// TIA Portal V15.1 export
// export: Created 2020-06-12T07:35:48.5224609Z, ExportSetting None, DisplayName Totally Integrated Automation Portal, DisplayVersion V15.1, DisplayName TIA Portal Openness, DisplayVersion V15.1, DisplayName STEP 7 Professional, DisplayVersion V15.1, DisplayName STEP 7 Safety, DisplayVersion V15.1, DisplayName WinCC Advanced, DisplayVersion V15.1
FUNCTION "PWR_trafo" : Void   // FC143, FBD
TITLE = Transformer with a vareing secondary voltage
{ S7_Optimized_Access := 'TRUE' }
// stored: SetENOAutomatically False
   VAR_TEMP
      tContEn : Bool;
      tContEnS : Bool;
      tContOn : Bool;
      tContLock : Bool;
      tContLStop : Bool;
      tContLSbot : Bool;
      tContCbOn : Bool;
      tContOnInc : Bool;
      tContOnDec : Bool;
      tContRunUp : Bool;
      tContRunDown : Bool;
      tOCTReq : Bool;
      tContMode : Int;
      tContSet : Real;   // Manipulation speed (cont K)
      tContFbSet : Real;
      tContUest : Real;   // Filtered actual voltage (filter K)
      tContUestS : Real;   // Filtered actual voltage (filter S)
      tContUact : Real;   // Unfiltered measured voltage
      tContUset : Real;   // Target voltage
      tContUmin : Real;   // Minimal voltage (w/o load)
      tContUmax : Real;   // Maximal voltage (w/o load)
      tContSmax : Real;   // Maximal speed setpoint
      tContSmin : Real;   // Minimal speed setpoint
      tContCycle : Time;
      tResult : Word;
      tTrafoCoolFault : Bool;
      tDirectOp : Bool;
      tTrdPosErr : LReal;
      tWindsPosErr : Real;
      tContIact : Real;
      tConMeasMode : Bool;
      tContUdrop : Real;
      tPosInv : Real;
      tContTgtReached : Bool;
      tXinternal : Real;
      tUload : Real;
      tIload : Real;
      tContUdrop2 : Real;
      tRbase : Real;
      tPosValid : Bool;
   END_VAR
BEGIN

REGION Network 1: Transformar is cooling
   // These signals are inverted
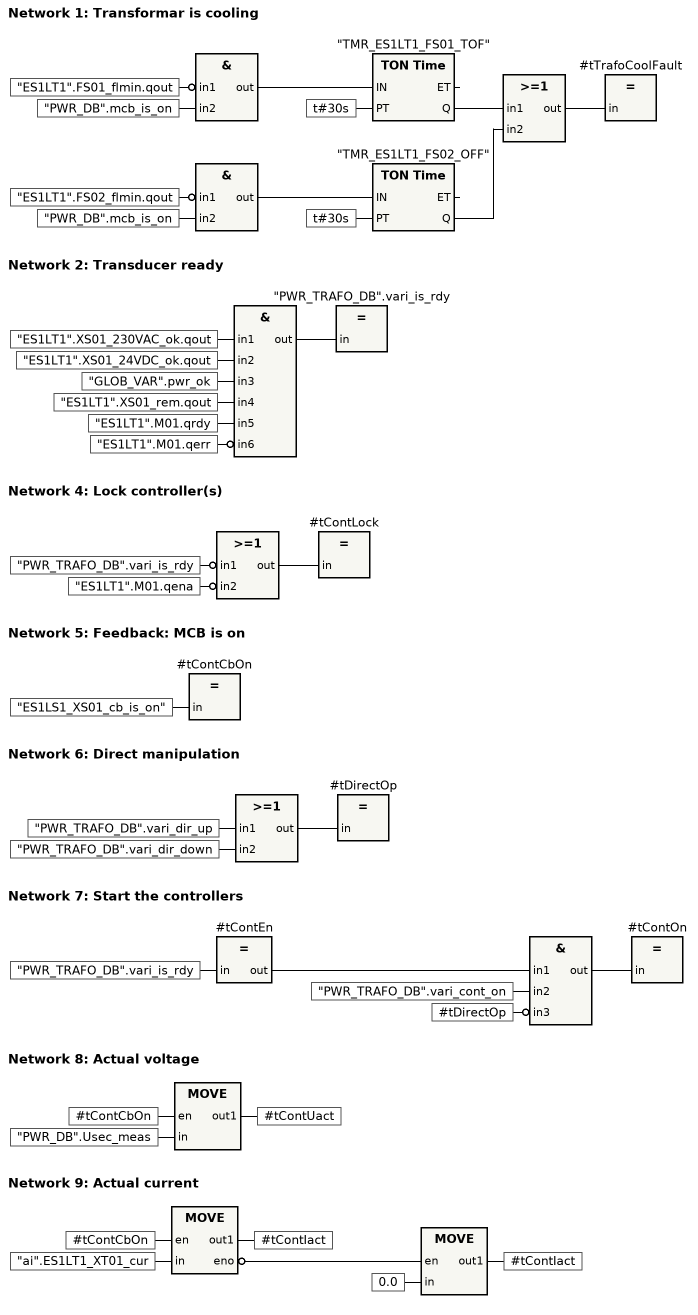
   "TMR_ES1LT1_FS01_TOF".TON(IN := NOT "ES1LT1".FS01_flmin.qout AND "PWR_DB".mcb_is_on, PT := t#30s);
   "TMR_ES1LT1_FS02_OFF".TON(IN := NOT "ES1LT1".FS02_flmin.qout AND "PWR_DB".mcb_is_on, PT := t#30s);
   #tTrafoCoolFault := "TMR_ES1LT1_FS01_TOF".Q OR "TMR_ES1LT1_FS02_OFF".Q;
END_REGION

REGION Network 2: Transducer ready
   "PWR_TRAFO_DB".vari_is_rdy := "ES1LT1".XS01_230VAC_ok.qout AND "ES1LT1".XS01_24VDC_ok.qout AND "GLOB_VAR".pwr_ok AND "ES1LT1".XS01_rem.qout AND "ES1LT1".M01.qrdy AND NOT "ES1LT1".M01.qerr;
END_REGION

REGION Network 3: -----------------------------------------------------------------------------
END_REGION

REGION Network 4: Lock controller(s)
   #tContLock := NOT "PWR_TRAFO_DB".vari_is_rdy OR NOT "ES1LT1".M01.qena;
END_REGION

REGION Network 5: Feedback: MCB is on
   #tContCbOn := "ES1LS1_XS01_cb_is_on";
END_REGION

REGION Network 6: Direct manipulation
   #tDirectOp := "PWR_TRAFO_DB".vari_dir_up OR "PWR_TRAFO_DB".vari_dir_down;
END_REGION

REGION Network 7: Start the controllers
   #tContEn := "PWR_TRAFO_DB".vari_is_rdy;
   #tContOn := "PWR_TRAFO_DB".vari_is_rdy AND "PWR_TRAFO_DB".vari_cont_on AND NOT #tDirectOp;
END_REGION

REGION Network 8: Actual voltage
   // I use these recalculation to avoid double model of voltage
   IF #tContCbOn THEN #tContUact := "PWR_DB".Usec_meas; END_IF;
END_REGION

REGION Network 9: Actual current
   IF #tContCbOn THEN #tContIact := "ai".ES1LT1_XT01_cur; END_IF;
   IF NOT #tContCbOn THEN #tContIact := 0.0; END_IF;
END_REGION

REGION Network 10: Measurement mode
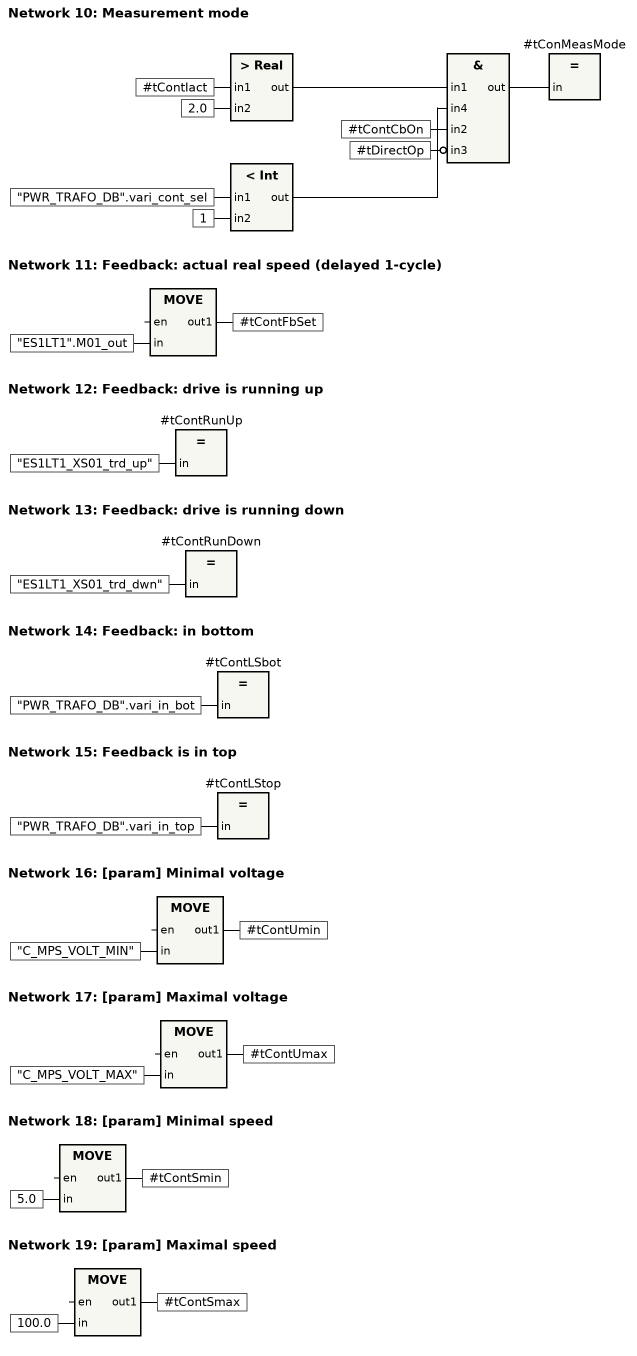
   #tConMeasMode := (#tContIact > 2.0) AND ("PWR_TRAFO_DB".vari_cont_sel < 1) AND #tContCbOn AND NOT #tDirectOp;
END_REGION

REGION Network 11: Feedback: actual real speed (delayed 1-cycle)
   #tContFbSet := "ES1LT1".M01_out;
END_REGION

REGION Network 12: Feedback: drive is running up
   #tContRunUp := "ES1LT1_XS01_trd_up";
END_REGION

REGION Network 13: Feedback: drive is running down
   #tContRunDown := "ES1LT1_XS01_trd_dwn";
END_REGION

REGION Network 14: Feedback: in bottom
   #tContLSbot := "PWR_TRAFO_DB".vari_in_bot;
END_REGION

REGION Network 15: Feedback is in top
   #tContLStop := "PWR_TRAFO_DB".vari_in_top;
END_REGION

REGION Network 16: [param] Minimal voltage
   #tContUmin := "C_MPS_VOLT_MIN";
END_REGION

REGION Network 17: [param] Maximal voltage
   #tContUmax := "C_MPS_VOLT_MAX";
END_REGION

REGION Network 18: [param] Minimal speed
   #tContSmin := 5.0;
END_REGION

REGION Network 19: [param] Maximal speed
   #tContSmax := 100.0;
END_REGION

REGION Network 20: [param] Cycle time
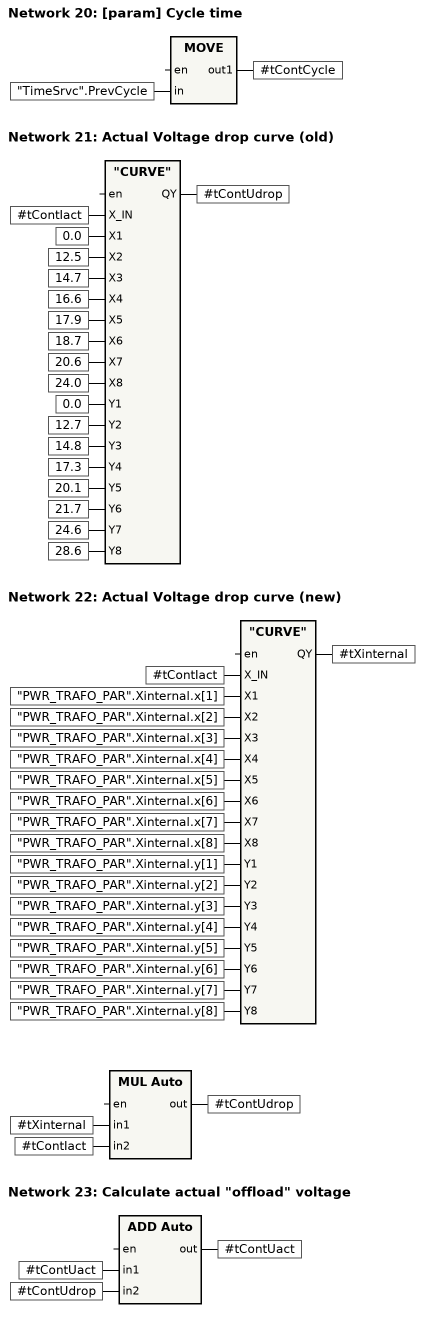
   #tContCycle := "TimeSrvc".PrevCycle;
END_REGION

REGION Network 21: Actual Voltage drop curve (old)
   // WARNING! After updating of the curve, you MUST update also the curve in the block FC "MELT_CPF_VP"
   "CURVE"(X_IN := #tContIact,
           X1 := 0.0,
           X2 := 12.5,
           X3 := 14.7,
           X4 := 16.6,
           X5 := 17.9,
           X6 := 18.7,
           X7 := 20.6,
           X8 := 24.0,
           Y1 := 0.0,
           Y2 := 12.7,
           Y3 := 14.8,
           Y4 := 17.3,
           Y5 := 20.1,
           Y6 := 21.7,
           Y7 := 24.6,
           Y8 := 28.6,
           QY => #tContUdrop);
END_REGION

REGION Network 22: Actual Voltage drop curve (new)
   // WARNING! After updating of the curve, you MUST update also the curve in the block FC "MELT_CPF_VP"
   "CURVE"(X_IN := #tContIact,
           X1 := "PWR_TRAFO_PAR".Xinternal.x[1],
           X2 := "PWR_TRAFO_PAR".Xinternal.x[2],
           X3 := "PWR_TRAFO_PAR".Xinternal.x[3],
           X4 := "PWR_TRAFO_PAR".Xinternal.x[4],
           X5 := "PWR_TRAFO_PAR".Xinternal.x[5],
           X6 := "PWR_TRAFO_PAR".Xinternal.x[6],
           X7 := "PWR_TRAFO_PAR".Xinternal.x[7],
           X8 := "PWR_TRAFO_PAR".Xinternal.x[8],
           Y1 := "PWR_TRAFO_PAR".Xinternal.y[1],
           Y2 := "PWR_TRAFO_PAR".Xinternal.y[2],
           Y3 := "PWR_TRAFO_PAR".Xinternal.y[3],
           Y4 := "PWR_TRAFO_PAR".Xinternal.y[4],
           Y5 := "PWR_TRAFO_PAR".Xinternal.y[5],
           Y6 := "PWR_TRAFO_PAR".Xinternal.y[6],
           Y7 := "PWR_TRAFO_PAR".Xinternal.y[7],
           Y8 := "PWR_TRAFO_PAR".Xinternal.y[8],
           QY => #tXinternal);
   #tContUdrop := #tXinternal * #tContIact;
END_REGION

REGION Network 23: Calculate actual "offload" voltage
   #tContUact := #tContUact + #tContUdrop;
END_REGION

REGION Network 24 (SCL): Calculate the resistance base
   IF "PWR_DB".current_flow THEN
       // I expect that this formula can do the power regulation a smooth
       #tRbase := 0.67 * "PWR_DB".Rsec_act + 0.33 * "PWR_DB".Rset;
       // but I am not sure. Well used old solution
       //#tRbase := "PWR_DB".Rsec_act;
   ELSE
       #tRbase := "PWR_DB".Rset;
   END_IF;
END_REGION

REGION Network 25: Calculate the voltage setpoint
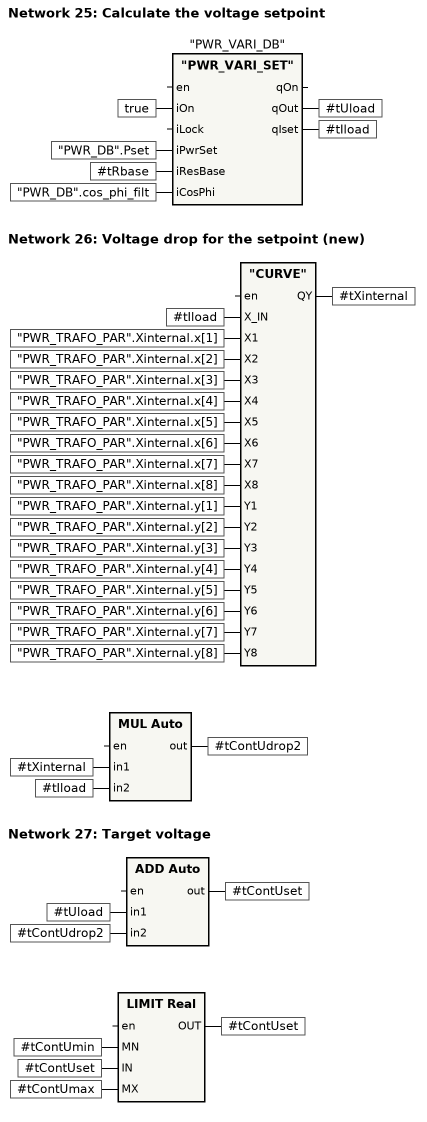
   "PWR_VARI_DB"(iOn := true,   // "PWR_VARI_SET"
                 iPwrSet := "PWR_DB".Pset,
                 iResBase := #tRbase,
                 iCosPhi := "PWR_DB".cos_phi_filt,
                 qOut => #tUload,
                 qIset => #tIload);
END_REGION

REGION Network 26: Voltage drop for the setpoint (new)
   "CURVE"(X_IN := #tIload,
           X1 := "PWR_TRAFO_PAR".Xinternal.x[1],
           X2 := "PWR_TRAFO_PAR".Xinternal.x[2],
           X3 := "PWR_TRAFO_PAR".Xinternal.x[3],
           X4 := "PWR_TRAFO_PAR".Xinternal.x[4],
           X5 := "PWR_TRAFO_PAR".Xinternal.x[5],
           X6 := "PWR_TRAFO_PAR".Xinternal.x[6],
           X7 := "PWR_TRAFO_PAR".Xinternal.x[7],
           X8 := "PWR_TRAFO_PAR".Xinternal.x[8],
           Y1 := "PWR_TRAFO_PAR".Xinternal.y[1],
           Y2 := "PWR_TRAFO_PAR".Xinternal.y[2],
           Y3 := "PWR_TRAFO_PAR".Xinternal.y[3],
           Y4 := "PWR_TRAFO_PAR".Xinternal.y[4],
           Y5 := "PWR_TRAFO_PAR".Xinternal.y[5],
           Y6 := "PWR_TRAFO_PAR".Xinternal.y[6],
           Y7 := "PWR_TRAFO_PAR".Xinternal.y[7],
           Y8 := "PWR_TRAFO_PAR".Xinternal.y[8],
           QY => #tXinternal);
   #tContUdrop2 := #tXinternal * #tIload;
END_REGION

REGION Network 27: Target voltage
   #tContUset := #tUload + #tContUdrop2;
   #tContUset := LIMIT(MN := #tContUmin, IN := #tContUset, MX := #tContUmax);
END_REGION

REGION Network 28: TRANSFORMER CONTROLLER
   // WARNING! The controler is VERY sensitive to the drive parameters
   // NOTE: 
   // - The bottom position of winds is a highest voltage
   // - The top position of winds is a lowest voltage
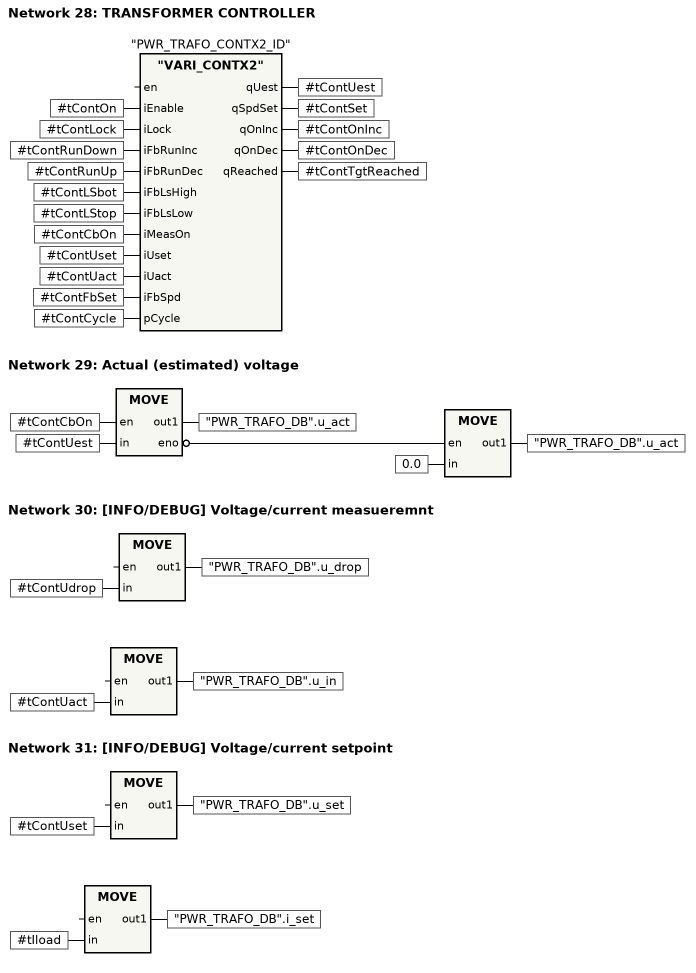
   "PWR_TRAFO_CONTX2_ID"(iEnable := #tContOn,   // "VARI_CONTX2"
                         iLock := #tContLock,
                         iFbRunInc := #tContRunDown,
                         iFbRunDec := #tContRunUp,
                         iFbLsHigh := #tContLSbot,
                         iFbLsLow := #tContLStop,
                         iMeasOn := #tContCbOn,
                         iUset := #tContUset,
                         iUact := #tContUact,
                         iFbSpd := #tContFbSet,
                         pCycle := #tContCycle,
                         qUest => #tContUest,
                         qSpdSet => #tContSet,
                         qOnInc => #tContOnInc,
                         qOnDec => #tContOnDec,
                         qReached => #tContTgtReached);
END_REGION

REGION Network 29: Actual (estimated) voltage
   IF #tContCbOn THEN "PWR_TRAFO_DB".u_act := #tContUest; END_IF;
   IF NOT #tContCbOn THEN "PWR_TRAFO_DB".u_act := 0.0; END_IF;
END_REGION

REGION Network 30: [INFO/DEBUG] Voltage/current measueremnt
   "PWR_TRAFO_DB".u_drop := #tContUdrop;
   "PWR_TRAFO_DB".u_in := #tContUact;
END_REGION

REGION Network 31: [INFO/DEBUG] Voltage/current setpoint
   "PWR_TRAFO_DB".u_set := #tContUset;
   "PWR_TRAFO_DB".i_set := #tIload;
END_REGION

REGION Network 32: [INFO/DEBUG] Voltage/current setpoint
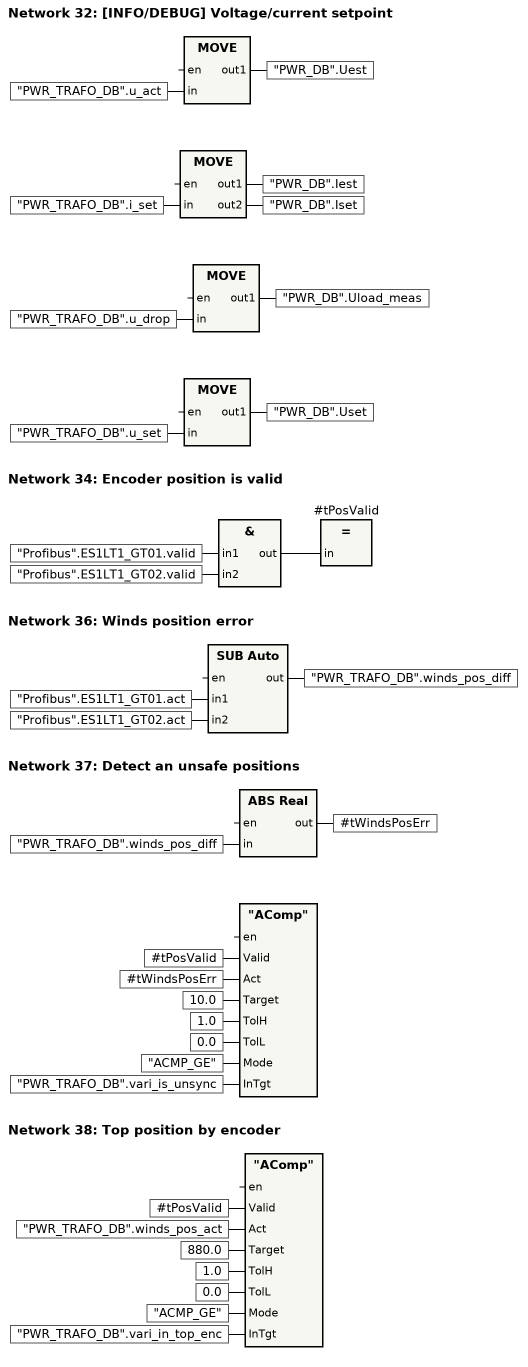
   "PWR_DB".Uest := "PWR_TRAFO_DB".u_act;
   "PWR_DB".Iest := "PWR_TRAFO_DB".i_set;
   "PWR_DB".Iset := "PWR_TRAFO_DB".i_set;
   "PWR_DB".Uload_meas := "PWR_TRAFO_DB".u_drop;
   "PWR_DB".Uset := "PWR_TRAFO_DB".u_set;
END_REGION

REGION Network 33: [Winds position]
END_REGION

REGION Network 34: Encoder position is valid
   #tPosValid := "Profibus".ES1LT1_GT01.valid AND "Profibus".ES1LT1_GT02.valid;
END_REGION

REGION Network 35 (SCL): Winds position calculation
   IF #tPosValid THEN
       "PWR_TRAFO_DB".winds_pos_act := 0.5 * ("Profibus".ES1LT1_GT01.act + "Profibus".ES1LT1_GT02.act);
   END_IF;
END_REGION

REGION Network 36: Winds position error
   "PWR_TRAFO_DB".winds_pos_diff := "Profibus".ES1LT1_GT01.act - "Profibus".ES1LT1_GT02.act;
END_REGION

REGION Network 37: Detect an unsafe positions
   #tWindsPosErr := ABS("PWR_TRAFO_DB".winds_pos_diff);
   "AComp"(Valid := #tPosValid,
           Act := #tWindsPosErr,
           Target := 10.0,
           TolH := 1.0,
           TolL := 0.0,
           Mode := "ACMP_GE",
           InTgt := "PWR_TRAFO_DB".vari_is_unsync);
END_REGION

REGION Network 38: Top position by encoder
   "AComp"(Valid := #tPosValid,
           Act := "PWR_TRAFO_DB".winds_pos_act,
           Target := 880.0,
           TolH := 1.0,
           TolL := 0.0,
           Mode := "ACMP_GE",
           InTgt := "PWR_TRAFO_DB".vari_in_top_enc);
END_REGION

REGION Network 39: Bottom position by encoder
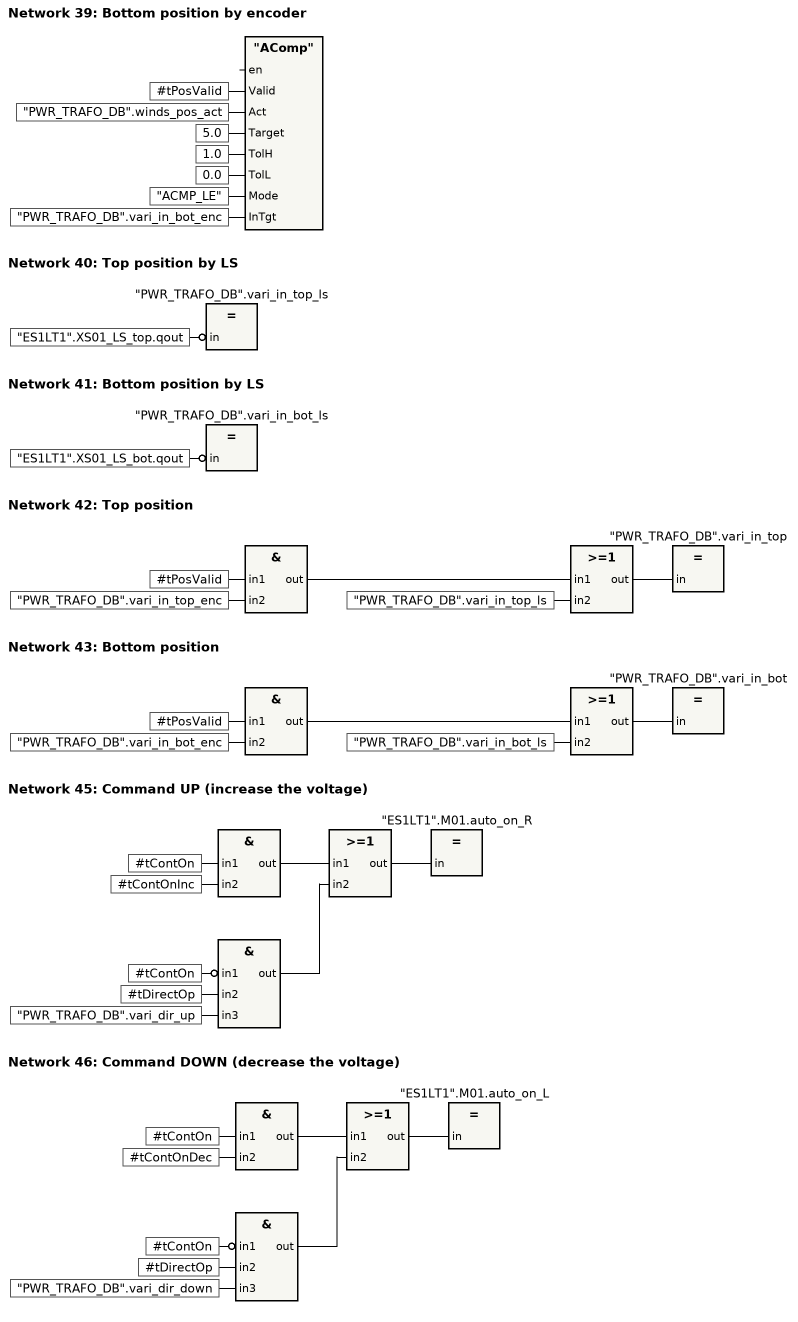
   "AComp"(Valid := #tPosValid,
           Act := "PWR_TRAFO_DB".winds_pos_act,
           Target := 5.0,
           TolH := 1.0,
           TolL := 0.0,
           Mode := "ACMP_LE",
           InTgt := "PWR_TRAFO_DB".vari_in_bot_enc);
END_REGION

REGION Network 40: Top position by LS
   "PWR_TRAFO_DB".vari_in_top_ls := NOT "ES1LT1".XS01_LS_top.qout;
END_REGION

REGION Network 41: Bottom position by LS
   "PWR_TRAFO_DB".vari_in_bot_ls := NOT "ES1LT1".XS01_LS_bot.qout;
END_REGION

REGION Network 42: Top position
   "PWR_TRAFO_DB".vari_in_top := (#tPosValid AND "PWR_TRAFO_DB".vari_in_top_enc) OR "PWR_TRAFO_DB".vari_in_top_ls;
END_REGION

REGION Network 43: Bottom position
   "PWR_TRAFO_DB".vari_in_bot := (#tPosValid AND "PWR_TRAFO_DB".vari_in_bot_enc) OR "PWR_TRAFO_DB".vari_in_bot_ls;
END_REGION

REGION Network 44: [Commands]
END_REGION

REGION Network 45: Command UP (increase the voltage)
   "ES1LT1".M01.auto_on_R := (#tContOn AND #tContOnInc) OR (NOT #tContOn AND #tDirectOp AND "PWR_TRAFO_DB".vari_dir_up);
END_REGION

REGION Network 46: Command DOWN (decrease the voltage)
   "ES1LT1".M01.auto_on_L := (#tContOn AND #tContOnDec) OR (NOT #tContOn AND #tDirectOp AND "PWR_TRAFO_DB".vari_dir_down);
END_REGION

REGION Network 47: Manipulation signal (drive speed)
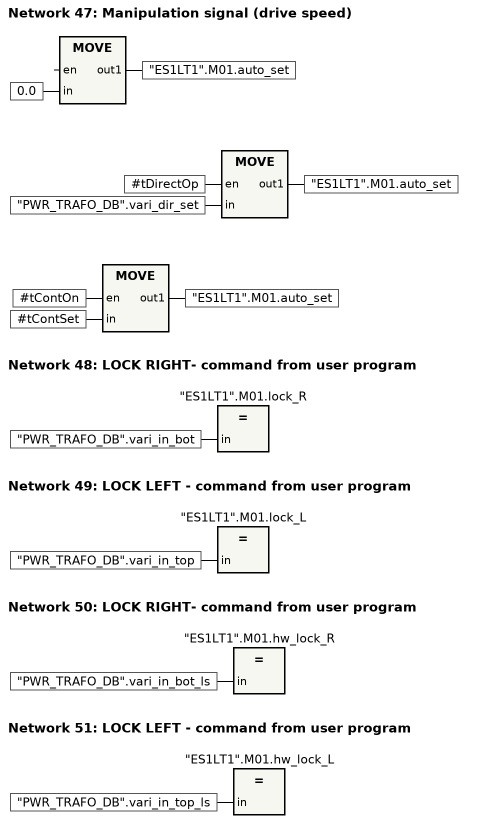
   "ES1LT1".M01.auto_set := 0.0;
   IF #tDirectOp THEN "ES1LT1".M01.auto_set := "PWR_TRAFO_DB".vari_dir_set; END_IF;
   IF #tContOn THEN "ES1LT1".M01.auto_set := #tContSet; END_IF;
END_REGION

REGION Network 48: LOCK RIGHT- command from user program
   "ES1LT1".M01.lock_R := "PWR_TRAFO_DB".vari_in_bot;
END_REGION

REGION Network 49: LOCK LEFT - command from user program
   "ES1LT1".M01.lock_L := "PWR_TRAFO_DB".vari_in_top;
END_REGION

REGION Network 50: LOCK RIGHT- command from user program
   "ES1LT1".M01.hw_lock_R := "PWR_TRAFO_DB".vari_in_bot_ls;
END_REGION

REGION Network 51: LOCK LEFT - command from user program
   "ES1LT1".M01.hw_lock_L := "PWR_TRAFO_DB".vari_in_top_ls;
END_REGION
END_FUNCTION
